    bool bActive
    bool bEnable = true
    dio dDio = {link=ApplicomIO-1\TOPIC1_A-BLOCKA\%Q48}
    string sID = "NetOut48"
    string sName = "NetOut48"
  [NetOut49]
    bool bActive
    bool bEnable = true
    dio dDio = {link=ApplicomIO-1\TOPIC1_A-BLOCKA\%Q49}
    string sID = "NetOut49"
    string sName = "NetOut49"
  [NetOut50]
    bool bActive
    bool bEnable = true
    dio dDio = {link=ApplicomIO-1\TOPIC1_A-BLOCKA\%Q50}
    string sID = "NetOut50"
    string sName = "NetOut50"
  [NetOut51]
    bool bActive
    bool bEnable = true
    dio dDio = {link=ApplicomIO-1\TOPIC1_A-BLOCKA\%Q51}
    string sID = "NetOut51"
    string sName = "NetOut51"
  [NetOut52]
    bool bActive
    bool bEnable = true
    dio dDio = {link=ApplicomIO-1\TOPIC1_A-BLOCKA\%Q52}
    string sID = "NetOut52"
    string sName = "NetOut52"
  [NetOut53]
    bool bActive
    bool bEnable = true
    dio dDio = {link=ApplicomIO-1\TOPIC1_A-BLOCKA\%Q53}
    string sID = "NetOut53"
    string sName = "NetOut53"
  [NetOut54]
    bool bActive
    bool bEnable = true
    dio dDio = {link=ApplicomIO-1\TOPIC1_A-BLOCKA\%Q54}
    string sID = "NetOut54"
    string sName = "NetOut54"
  [NetOut55]
    bool bActive
    bool bEnable = true
    dio dDio = {link=ApplicomIO-1\TOPIC1_A-BLOCKA\%Q55}
    string sID = "NetOut55"
    string sName = "NetOut55"
  [NetOut56]
    bool bActive
    bool bEnable = true
    dio dDio = {link=ApplicomIO-1\TOPIC1_A-BLOCKA\%Q56}
    string sID = "NetOut56"
    string sName = "NetOut56"
  [NetOut57]
    bool bActive
    bool bEnable = true
    dio dDio = {link=ApplicomIO-1\TOPIC1_A-BLOCKA\%Q57}
    string sID = "NetOut57"
    string sName = "NetOut57"
  [NetOut58]
    bool bActive
    bool bEnable = true
    dio dDio = {link=ApplicomIO-1\TOPIC1_A-BLOCKA\%Q58}
    string sID = "NetOut58"
    string sName = "NetOut58"
  [NetOut59]
    bool bActive
    bool bEnable = true
    dio dDio = {link=ApplicomIO-1\TOPIC1_A-BLOCKA\%Q59}
    string sID = "NetOut59"
    string sName = "NetOut59"
  [NetOut60]
    bool bActive
    bool bEnable = true
    dio dDio = {link=ApplicomIO-1\TOPIC1_A-BLOCKA\%Q60}
    string sID = "NetOut60"
    string sName = "NetOut60"
  [NetOut61]
    bool bActive
    bool bEnable = true
    dio dDio = {link=ApplicomIO-1\TOPIC1_A-BLOCKA\%Q61}
    string sID = "NetOut61"
    string sName = "NetOut61"
  [NetOut62]
    bool bActive
    bool bEnable = true
    dio dDio = {link=ApplicomIO-1\TOPIC1_A-BLOCKA\%Q62}
    string sID = "NetOut62"
    string sName = "NetOut62"
  [NetOut63]
    bool bActive
    bool bEnable = true
    dio dDio = {link=ApplicomIO-1\TOPIC1_A-BLOCKA\%Q63}
    string sID = "NetOut63"
    string sName = "NetOut63"
  [fOut0]
    bool bActive = true
    bool bEnable = true
    dio dDio = {link=fOut0}
    string sID = "fOut0"
    string sName = "fOut0"
  [valve1]
    bool bActive = true
    bool bEnable = true
    dio dDio = {link=valve1}
    string sID = "valve1"
    string sName = "valve1"
  [valve2]
    bool bActive = true
    bool bEnable = true
    dio dDio = {link=valve2}
    string sID = "valve2"
    string sName = "valve2"
public num nCounter[10]
public string sCondition[6]
  [0] = "!="
  [1] = ">="
  [2] = "> "
  [3] = "< "
  [4] = "<="
  [5] = "=="
public string sOperator[4]
  [0] = "= "
  [1] = "=NUM "
  [2] = "+1"
  [3] = "-1"
